FUNCTION_BLOCK Call_Fb
VAR_INPUT
END_VAR
VAR_OUTPUT
END_VAR
VAR
	Feedback_CC1_Clamp1: Feedback;
	Feedback_CC1_Clamp2: Feedback;
	Feedback_CC1_Clamp3: Feedback;
	Feedback_CC2_Clamp1: Feedback;
	Feedback_CC2_Clamp2: Feedback;
	Feedback_CC2_Clamp3: Feedback;
	Feedback_CC3_Clamp1: Feedback;
	Feedback_CC3_Clamp2: Feedback;
	Feedback_CC3_Clamp3: Feedback;
	Feedback_CC4_Clamp1: Feedback;
	Feedback_CC4_Clamp2: Feedback;
	Feedback_CC4_Clamp3: Feedback;
	Feedback_CC5_Clamp1: Feedback;
	Feedback_CC6_Clamp1: Feedback;

	Feedback_TT: Feedback;
	Feedback_TT1: Feedback;
	Turn_Table_0: Turn_Table;

		Turning_fb_0: Turning_fb;
	Feedback_Turn: Feedback;
	Feedback_Turn1: Feedback;
	RoolerDoor_1: RoolerDoor;
	Feedback_RD1: Feedback;
	RoolerDoor_2: RoolerDoor;
	Feedback_RD2: Feedback;
	Robot_MH: RobotMH;
	AutoSequence_0: AutoSequence;
	WeldRobot_0: WeldRobot;
	
END_VAR

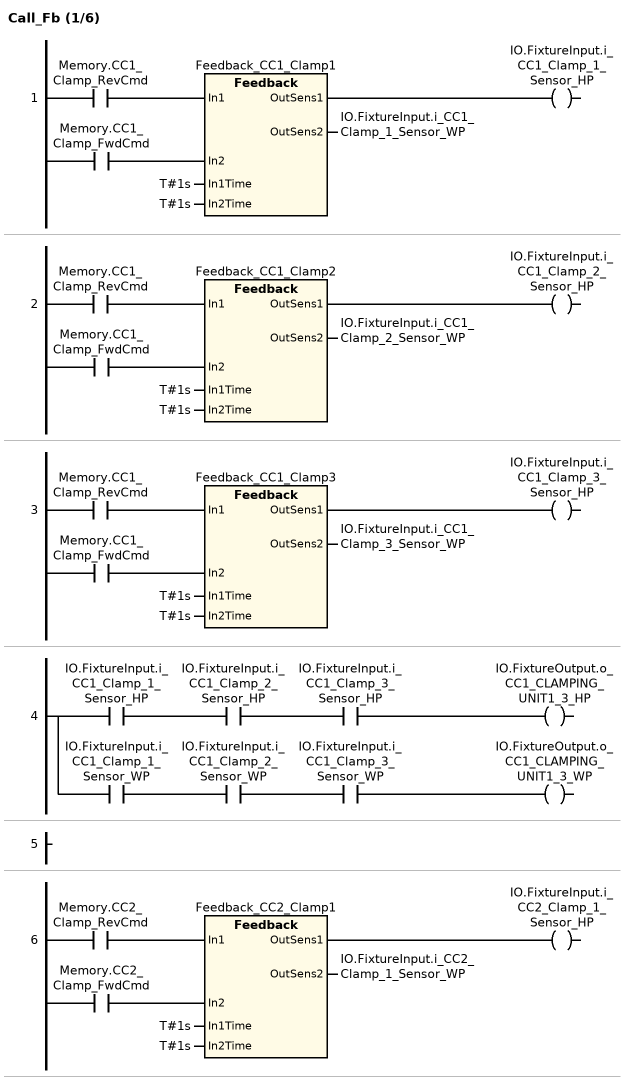
// NETWORK 1
Feedback_CC1_Clamp1(
    In1 := Memory.CC1_Clamp_RevCmd,
    In2 := Memory.CC1_Clamp_FwdCmd,
    In1Time := T#1s,
    In2Time := T#1s,
    OutSens2 => IO.FixtureInput.i_CC1_Clamp_1_Sensor_WP); // Feedback
IO.FixtureInput.i_CC1_Clamp_1_Sensor_HP := Feedback_CC1_Clamp1.OutSens1;

// NETWORK 2
Feedback_CC1_Clamp2(
    In1 := Memory.CC1_Clamp_RevCmd,
    In2 := Memory.CC1_Clamp_FwdCmd,
    In1Time := T#1s,
    In2Time := T#1s,
    OutSens2 => IO.FixtureInput.i_CC1_Clamp_2_Sensor_WP); // Feedback
IO.FixtureInput.i_CC1_Clamp_2_Sensor_HP := Feedback_CC1_Clamp2.OutSens1;

// NETWORK 3
Feedback_CC1_Clamp3(
    In1 := Memory.CC1_Clamp_RevCmd,
    In2 := Memory.CC1_Clamp_FwdCmd,
    In1Time := T#1s,
    In2Time := T#1s,
    OutSens2 => IO.FixtureInput.i_CC1_Clamp_3_Sensor_WP); // Feedback
IO.FixtureInput.i_CC1_Clamp_3_Sensor_HP := Feedback_CC1_Clamp3.OutSens1;

// NETWORK 4
IO.FixtureOutput.o_CC1_CLAMPING_UNIT1_3_HP := IO.FixtureInput.i_CC1_Clamp_1_Sensor_HP AND IO.FixtureInput.i_CC1_Clamp_2_Sensor_HP AND IO.FixtureInput.i_CC1_Clamp_3_Sensor_HP;
IO.FixtureOutput.o_CC1_CLAMPING_UNIT1_3_WP := IO.FixtureInput.i_CC1_Clamp_1_Sensor_WP AND IO.FixtureInput.i_CC1_Clamp_2_Sensor_WP AND IO.FixtureInput.i_CC1_Clamp_3_Sensor_WP;

// NETWORK 5

// NETWORK 6
Feedback_CC2_Clamp1(
    In1 := Memory.CC2_Clamp_RevCmd,
    In2 := Memory.CC2_Clamp_FwdCmd,
    In1Time := T#1s,
    In2Time := T#1s,
    OutSens2 => IO.FixtureInput.i_CC2_Clamp_1_Sensor_WP); // Feedback
IO.FixtureInput.i_CC2_Clamp_1_Sensor_HP := Feedback_CC2_Clamp1.OutSens1;

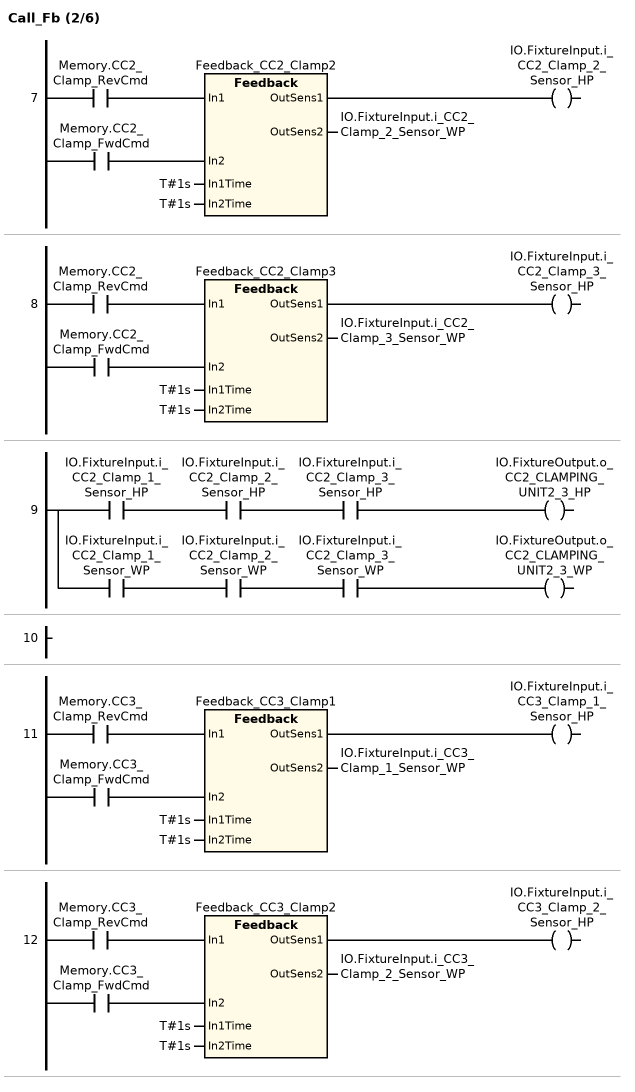
// NETWORK 7
Feedback_CC2_Clamp2(
    In1 := Memory.CC2_Clamp_RevCmd,
    In2 := Memory.CC2_Clamp_FwdCmd,
    In1Time := T#1s,
    In2Time := T#1s,
    OutSens2 => IO.FixtureInput.i_CC2_Clamp_2_Sensor_WP); // Feedback
IO.FixtureInput.i_CC2_Clamp_2_Sensor_HP := Feedback_CC2_Clamp2.OutSens1;

// NETWORK 8
Feedback_CC2_Clamp3(
    In1 := Memory.CC2_Clamp_RevCmd,
    In2 := Memory.CC2_Clamp_FwdCmd,
    In1Time := T#1s,
    In2Time := T#1s,
    OutSens2 => IO.FixtureInput.i_CC2_Clamp_3_Sensor_WP); // Feedback
IO.FixtureInput.i_CC2_Clamp_3_Sensor_HP := Feedback_CC2_Clamp3.OutSens1;

// NETWORK 9
IO.FixtureOutput.o_CC2_CLAMPING_UNIT2_3_HP := IO.FixtureInput.i_CC2_Clamp_1_Sensor_HP AND IO.FixtureInput.i_CC2_Clamp_2_Sensor_HP AND IO.FixtureInput.i_CC2_Clamp_3_Sensor_HP;
IO.FixtureOutput.o_CC2_CLAMPING_UNIT2_3_WP := IO.FixtureInput.i_CC2_Clamp_1_Sensor_WP AND IO.FixtureInput.i_CC2_Clamp_2_Sensor_WP AND IO.FixtureInput.i_CC2_Clamp_3_Sensor_WP;

// NETWORK 10

// NETWORK 11
Feedback_CC3_Clamp1(
    In1 := Memory.CC3_Clamp_RevCmd,
    In2 := Memory.CC3_Clamp_FwdCmd,
    In1Time := T#1s,
    In2Time := T#1s,
    OutSens2 => IO.FixtureInput.i_CC3_Clamp_1_Sensor_WP); // Feedback
IO.FixtureInput.i_CC3_Clamp_1_Sensor_HP := Feedback_CC3_Clamp1.OutSens1;

// NETWORK 12
Feedback_CC3_Clamp2(
    In1 := Memory.CC3_Clamp_RevCmd,
    In2 := Memory.CC3_Clamp_FwdCmd,
    In1Time := T#1s,
    In2Time := T#1s,
    OutSens2 => IO.FixtureInput.i_CC3_Clamp_2_Sensor_WP); // Feedback
IO.FixtureInput.i_CC3_Clamp_2_Sensor_HP := Feedback_CC3_Clamp2.OutSens1;

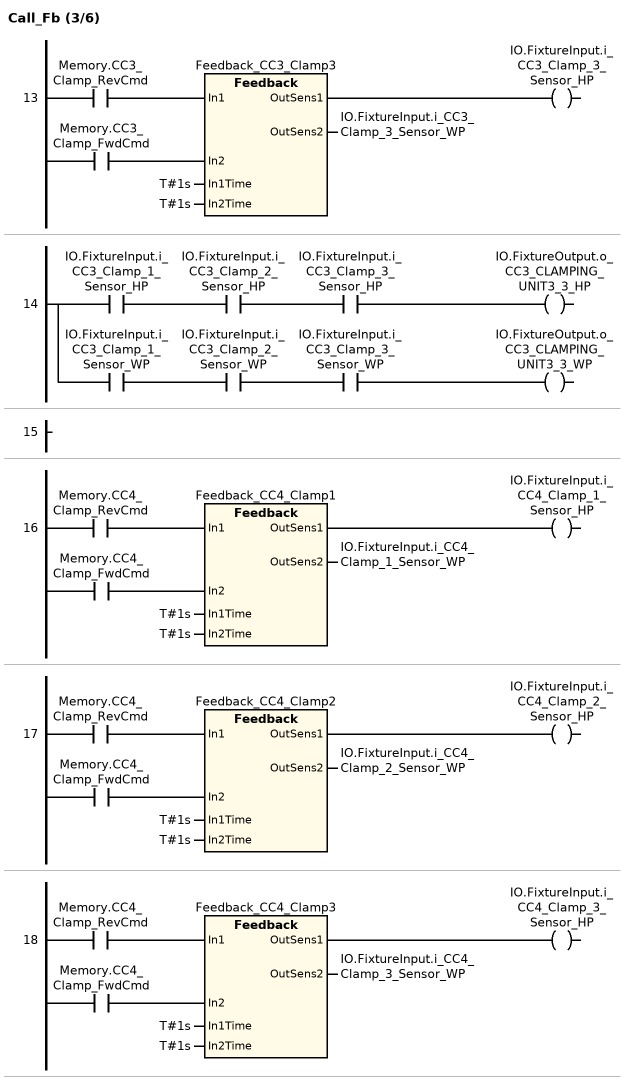
// NETWORK 13
Feedback_CC3_Clamp3(
    In1 := Memory.CC3_Clamp_RevCmd,
    In2 := Memory.CC3_Clamp_FwdCmd,
    In1Time := T#1s,
    In2Time := T#1s,
    OutSens2 => IO.FixtureInput.i_CC3_Clamp_3_Sensor_WP); // Feedback
IO.FixtureInput.i_CC3_Clamp_3_Sensor_HP := Feedback_CC3_Clamp3.OutSens1;

// NETWORK 14
IO.FixtureOutput.o_CC3_CLAMPING_UNIT3_3_HP := IO.FixtureInput.i_CC3_Clamp_1_Sensor_HP AND IO.FixtureInput.i_CC3_Clamp_2_Sensor_HP AND IO.FixtureInput.i_CC3_Clamp_3_Sensor_HP;
IO.FixtureOutput.o_CC3_CLAMPING_UNIT3_3_WP := IO.FixtureInput.i_CC3_Clamp_1_Sensor_WP AND IO.FixtureInput.i_CC3_Clamp_2_Sensor_WP AND IO.FixtureInput.i_CC3_Clamp_3_Sensor_WP;

// NETWORK 15

// NETWORK 16
Feedback_CC4_Clamp1(
    In1 := Memory.CC4_Clamp_RevCmd,
    In2 := Memory.CC4_Clamp_FwdCmd,
    In1Time := T#1s,
    In2Time := T#1s,
    OutSens2 => IO.FixtureInput.i_CC4_Clamp_1_Sensor_WP); // Feedback
IO.FixtureInput.i_CC4_Clamp_1_Sensor_HP := Feedback_CC4_Clamp1.OutSens1;

// NETWORK 17
Feedback_CC4_Clamp2(
    In1 := Memory.CC4_Clamp_RevCmd,
    In2 := Memory.CC4_Clamp_FwdCmd,
    In1Time := T#1s,
    In2Time := T#1s,
    OutSens2 => IO.FixtureInput.i_CC4_Clamp_2_Sensor_WP); // Feedback
IO.FixtureInput.i_CC4_Clamp_2_Sensor_HP := Feedback_CC4_Clamp2.OutSens1;

// NETWORK 18
Feedback_CC4_Clamp3(
    In1 := Memory.CC4_Clamp_RevCmd,
    In2 := Memory.CC4_Clamp_FwdCmd,
    In1Time := T#1s,
    In2Time := T#1s,
    OutSens2 => IO.FixtureInput.i_CC4_Clamp_3_Sensor_WP); // Feedback
IO.FixtureInput.i_CC4_Clamp_3_Sensor_HP := Feedback_CC4_Clamp3.OutSens1;

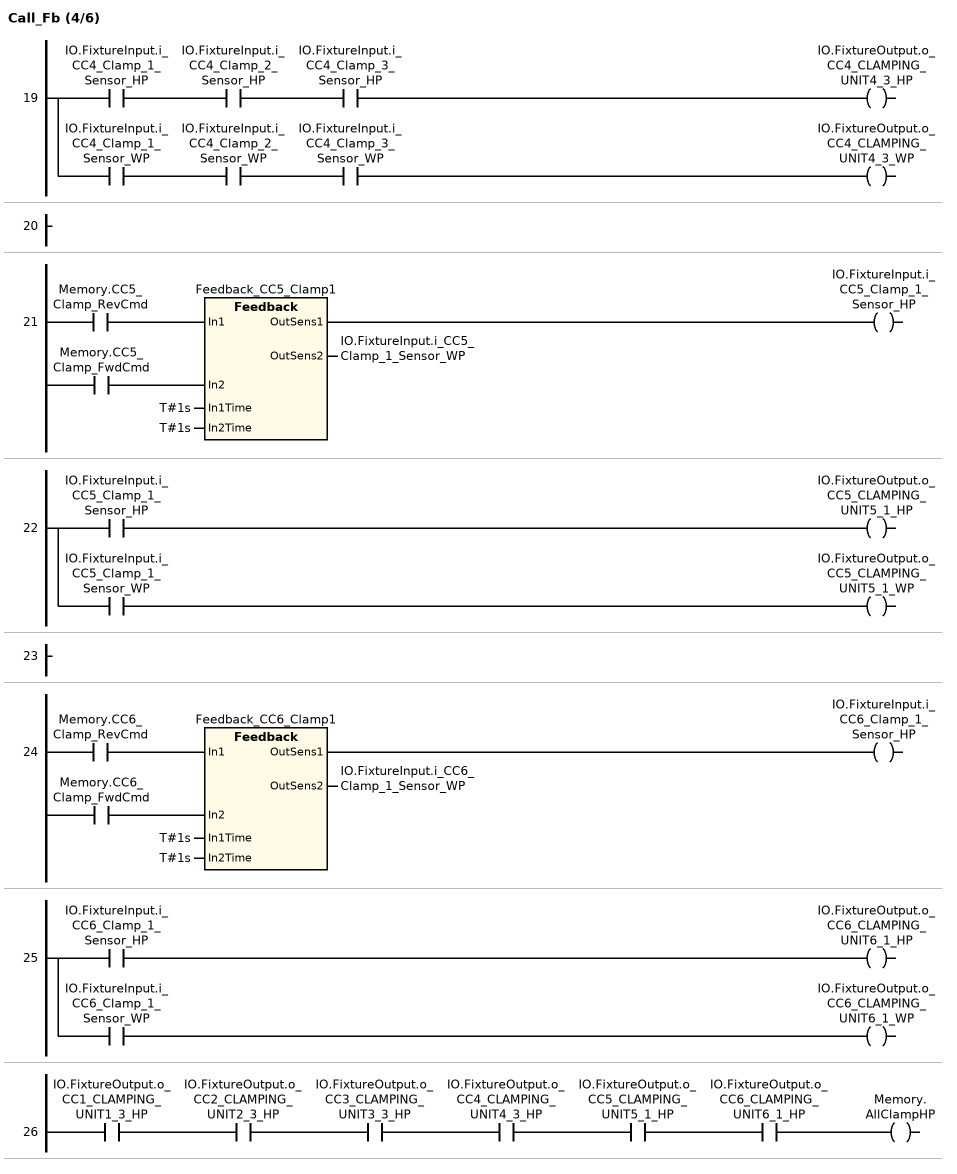
// NETWORK 19
IO.FixtureOutput.o_CC4_CLAMPING_UNIT4_3_HP := IO.FixtureInput.i_CC4_Clamp_1_Sensor_HP AND IO.FixtureInput.i_CC4_Clamp_2_Sensor_HP AND IO.FixtureInput.i_CC4_Clamp_3_Sensor_HP;
IO.FixtureOutput.o_CC4_CLAMPING_UNIT4_3_WP := IO.FixtureInput.i_CC4_Clamp_1_Sensor_WP AND IO.FixtureInput.i_CC4_Clamp_2_Sensor_WP AND IO.FixtureInput.i_CC4_Clamp_3_Sensor_WP;

// NETWORK 20

// NETWORK 21
Feedback_CC5_Clamp1(
    In1 := Memory.CC5_Clamp_RevCmd,
    In2 := Memory.CC5_Clamp_FwdCmd,
    In1Time := T#1s,
    In2Time := T#1s,
    OutSens2 => IO.FixtureInput.i_CC5_Clamp_1_Sensor_WP); // Feedback
IO.FixtureInput.i_CC5_Clamp_1_Sensor_HP := Feedback_CC5_Clamp1.OutSens1;

// NETWORK 22
IO.FixtureOutput.o_CC5_CLAMPING_UNIT5_1_HP := IO.FixtureInput.i_CC5_Clamp_1_Sensor_HP;
IO.FixtureOutput.o_CC5_CLAMPING_UNIT5_1_WP := IO.FixtureInput.i_CC5_Clamp_1_Sensor_WP;

// NETWORK 23

// NETWORK 24
Feedback_CC6_Clamp1(
    In1 := Memory.CC6_Clamp_RevCmd,
    In2 := Memory.CC6_Clamp_FwdCmd,
    In1Time := T#1s,
    In2Time := T#1s,
    OutSens2 => IO.FixtureInput.i_CC6_Clamp_1_Sensor_WP); // Feedback
IO.FixtureInput.i_CC6_Clamp_1_Sensor_HP := Feedback_CC6_Clamp1.OutSens1;

// NETWORK 25
IO.FixtureOutput.o_CC6_CLAMPING_UNIT6_1_HP := IO.FixtureInput.i_CC6_Clamp_1_Sensor_HP;
IO.FixtureOutput.o_CC6_CLAMPING_UNIT6_1_WP := IO.FixtureInput.i_CC6_Clamp_1_Sensor_WP;

// NETWORK 26
Memory.AllClampHP := IO.FixtureOutput.o_CC1_CLAMPING_UNIT1_3_HP AND IO.FixtureOutput.o_CC2_CLAMPING_UNIT2_3_HP AND IO.FixtureOutput.o_CC3_CLAMPING_UNIT3_3_HP AND IO.FixtureOutput.o_CC4_CLAMPING_UNIT4_3_HP AND IO.FixtureOutput.o_CC5_CLAMPING_UNIT5_1_HP AND IO.FixtureOutput.o_CC6_CLAMPING_UNIT6_1_HP;

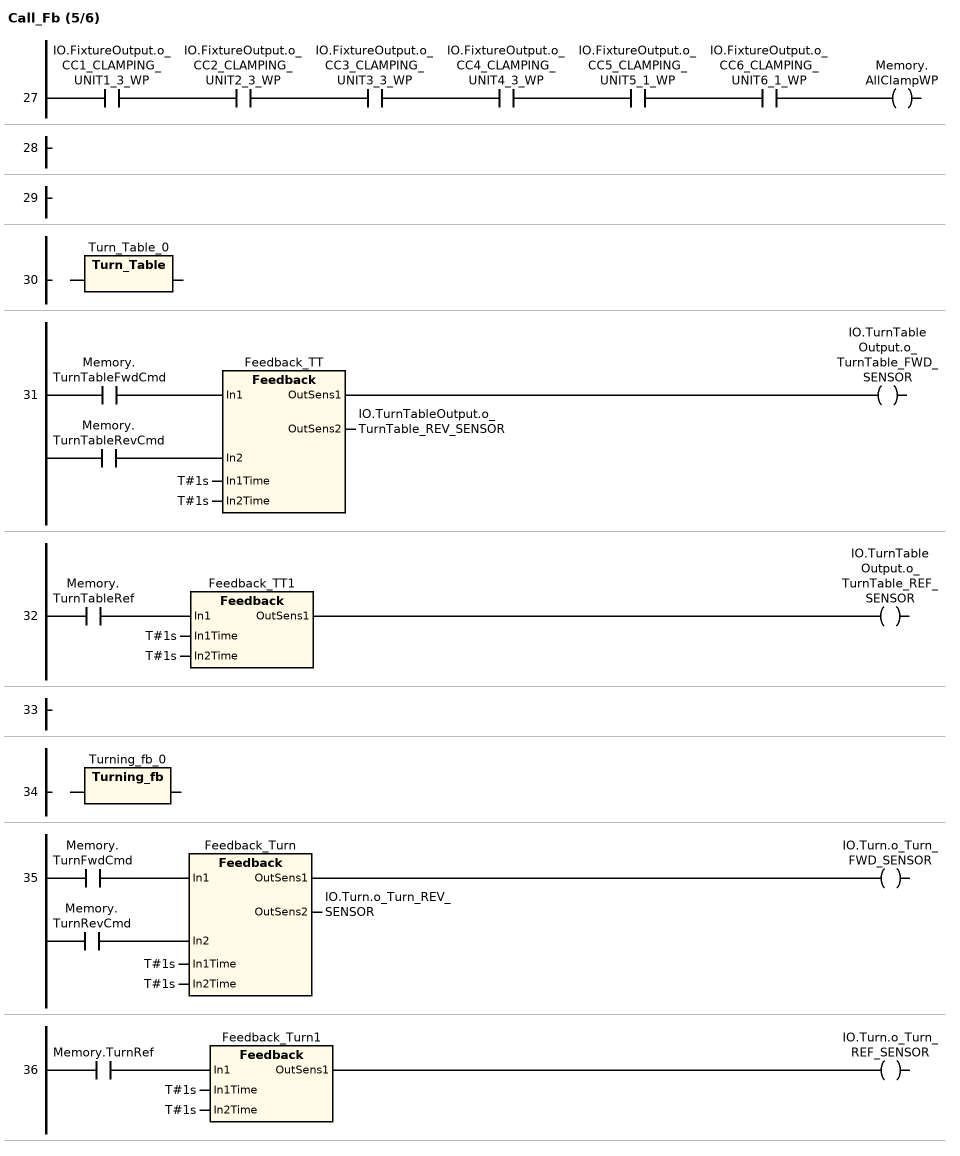
// NETWORK 27
Memory.AllClampWP := IO.FixtureOutput.o_CC1_CLAMPING_UNIT1_3_WP AND IO.FixtureOutput.o_CC2_CLAMPING_UNIT2_3_WP AND IO.FixtureOutput.o_CC3_CLAMPING_UNIT3_3_WP AND IO.FixtureOutput.o_CC4_CLAMPING_UNIT4_3_WP AND IO.FixtureOutput.o_CC5_CLAMPING_UNIT5_1_WP AND IO.FixtureOutput.o_CC6_CLAMPING_UNIT6_1_WP;

// NETWORK 28

// NETWORK 29

// NETWORK 30
Turn_Table_0(); // Turn_Table

// NETWORK 31
Feedback_TT(
    In1 := Memory.TurnTableFwdCmd,
    In2 := Memory.TurnTableRevCmd,
    In1Time := T#1s,
    In2Time := T#1s,
    OutSens2 => IO.TurnTableOutput.o_TurnTable_REV_SENSOR); // Feedback
IO.TurnTableOutput.o_TurnTable_FWD_SENSOR := Feedback_TT.OutSens1;

// NETWORK 32
Feedback_TT1(In1 := Memory.TurnTableRef, In1Time := T#1s, In2Time := T#1s); // Feedback
IO.TurnTableOutput.o_TurnTable_REF_SENSOR := Feedback_TT1.OutSens1;

// NETWORK 33

// NETWORK 34
Turning_fb_0(); // Turning_fb

// NETWORK 35
Feedback_Turn(
    In1 := Memory.TurnFwdCmd,
    In2 := Memory.TurnRevCmd,
    In1Time := T#1s,
    In2Time := T#1s,
    OutSens2 => IO.Turn.o_Turn_REV_SENSOR); // Feedback
IO.Turn.o_Turn_FWD_SENSOR := Feedback_Turn.OutSens1;

// NETWORK 36
Feedback_Turn1(In1 := Memory.TurnRef, In1Time := T#1s, In2Time := T#1s); // Feedback
IO.Turn.o_Turn_REF_SENSOR := Feedback_Turn1.OutSens1;

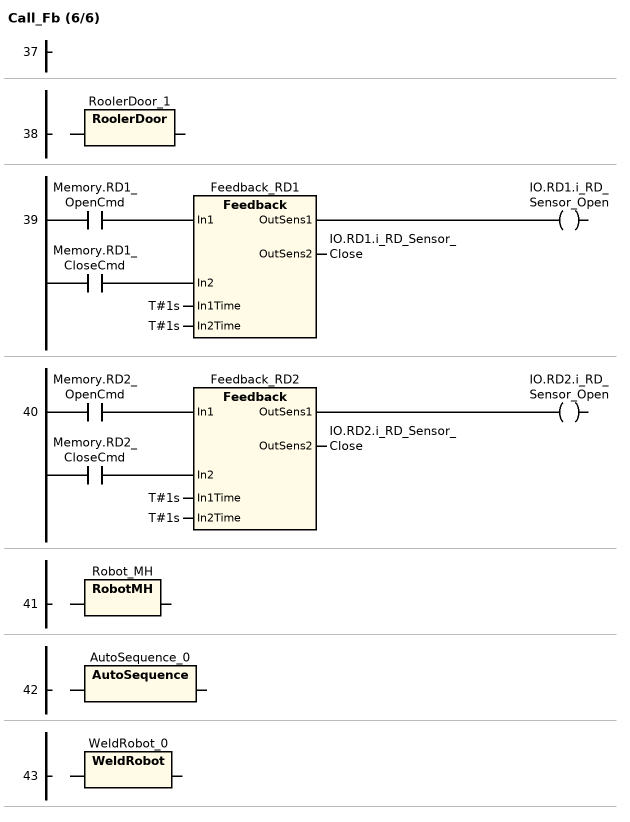
// NETWORK 37

// NETWORK 38
RoolerDoor_1(); // RoolerDoor

// NETWORK 39
Feedback_RD1(
    In1 := Memory.RD1_OpenCmd,
    In2 := Memory.RD1_CloseCmd,
    In1Time := T#1s,
    In2Time := T#1s,
    OutSens2 => IO.RD1.i_RD_Sensor_Close); // Feedback
IO.RD1.i_RD_Sensor_Open := Feedback_RD1.OutSens1;

// NETWORK 40
Feedback_RD2(
    In1 := Memory.RD2_OpenCmd,
    In2 := Memory.RD2_CloseCmd,
    In1Time := T#1s,
    In2Time := T#1s,
    OutSens2 => IO.RD2.i_RD_Sensor_Close); // Feedback
IO.RD2.i_RD_Sensor_Open := Feedback_RD2.OutSens1;

// NETWORK 41
Robot_MH(); // RobotMH

// NETWORK 42
AutoSequence_0(); // AutoSequence

// NETWORK 43
WeldRobot_0(); // WeldRobot

END_FUNCTION_BLOCK

(* stored: Version 1.1.0.1, ProductVersion 3.1.4024.16
   POU Call_Fb: Id {3e04f3c8-c02c-4594-8b2e-1834804af45a}, SpecialFunc None *)
